   MachineConfig[11]."Unknown"."EM - 463"."PIT463-1".CW.ENABLE := True;

   MachineConfig[11]."Unit Sep"."EM - 400"."FIT409-1".CW.ENABLE := True;

   MachineConfig[11]."Unit Process"."EM - 201"."FCV201-1".CW.EXIST := False;

   MachineConfig[11]."Unit Process"."EM - 22X"."PCV22X-1".CW.NO := True;

   MachineConfig[11]."Unit Process"."EM - 22Y"."PCV22Y-1".CW.EXIST := False;

   MachineConfig[11]."Unit Sep"."EM - 400"."FCV409-1".CW.ENABLE := True;

   MachineConfig[11]."Unit Sep"."EM - 100".UPS.CW.EXIST := True;

   MachineConfig[11]."Unit Sep"."EM - 730".TS730.CW.ENABLE := True;

   MachineConfig[11]."Unit Dch"."EM - 222"."LS222-1".CW.EXIST := False;

   MachineConfig[11]."Unit Dch"."EM - 222"."P222-1".CW.EXIST := False;

   MachineConfig[11]."Unknown"."EM - 420"."P403-1".CW.EXIST := False;

   MachineConfig[11]."Unknown"."EM - 430"."P406-1".CW.EXIST := False;

   MachineConfig[11]."Unknown"."EM - 463"."P463-1".CW.ENABLE := True;

   MachineConfig[11]."Unknown"."EM - 463"."P463-1".CW.EXIST := False;

   MachineConfig[11]."Options"."EM - P201"."P201-1".CW.EXIST := False;

   MachineConfig[11]."Unknown"."EM - 208"."P208-1".CW.EXIST := False;

   MachineConfig[11]."Unit Sep"."EM - 100"."CA ERROR".CW.NO := True;

   MachineConfig[11]."Unit Sep"."EM - 100"."CA WD".CW.NO := True;

   MachineConfig[11]."Unit Sep"."EM - 400"."FIS412-1".CW.EXIST := False;

   MachineConfig[11]."Unknown"."EM - 420".LS422a.CW.EXIST := False;

   MachineConfig[11]."Unknown"."EM - 420"."LS42X(b)".CW.EXIST := False;

   MachineConfig[11]."Unknown"."EM - 420"."LS422-1".CW.EXIST := False;

   MachineConfig[11]."Unit Sep"."EM - 400"."FIT412-1".CW.EXIST := False;

   MachineConfig[11]."Unit Dch"."EM - 375"."PT37X-1".CW.ENABLE := True;

   MachineConfig[11]."Unit Dch"."EM - 375"."PT37X-1".CW.EXIST := False;

   MachineConfig[11]."Unit Dch"."EM - 222"."TT222-1".CW.ENABLE := True;

   MachineConfig[11]."Unit Sep"."EM - 400"."TT411-1".CW.EXIST := False;

   MachineConfig[11]."Unit Sep"."EM - 730".TT730b.CW.EXIST := False;

   MachineConfig[11]."Unit Sep"."EM - 730".TT734.CW.EXIST := False;

   MachineConfig[11]."Unit Sep"."EM - 400"."TT41X-1".CW.ENABLE := True;

   MachineConfig[11]."Unit Dch"."EM - 300"."AV302-1".CW.EXIST := False;

   MachineConfig[11]."Unit Dch"."EM - 300"."AV303-1".CW.ENABLE := True;

   MachineConfig[11]."Unit Dch"."EM - 300"."AV304-1".CW.ENABLE := True;

   MachineConfig[11]."Unit Dch"."EM - 300"."AV305-1".CW.ENABLE := True;

   MachineConfig[11]."Unit Dch"."EM - 300"."AV306-1".CW.EXIST := False;

   MachineConfig[11]."Unit Sep"."EM - 600"."AV615-1".CW.ENABLE := True;

   MachineConfig[11]."Unit Dch"."EM - 300"."AV635-1".CW.ENABLE := True;

   MachineConfig[11]."Unit Sep"."EM - 600"."AV63X/441-1".CW.EXIST := False;

   MachineConfig[11]."Unknown"."EM - 420"."PV421-1".CW.EXIST := False;

   MachineConfig[11]."Unknown"."EM - 420"."P421-1".CW.EXIST := False;

   MachineConfig[11]."Unit Dch"."EM - 506"."PV376-1".CW.ENABLE := True;

   MachineConfig[11]."Unit Dch"."EM - 506"."PV376-1".CW.EXIST := False;

   MachineConfig[11]."Unit Dch"."EM - 506"."PV376-2".CW.ENABLE := True;

   MachineConfig[11]."Unit Dch"."EM - 506"."PV376-2".CW.EXIST := False;

   MachineConfig[11]."Unit Dch"."EM - 506"."PV376-2".CW.NO := True;

   MachineConfig[11]."Unknown"."EM - 463"."AV660-1".CW.ENABLE := True;

   MachineConfig[11]."Unknown"."EM - 463"."AV660-1".CW.EXIST := False;

   MachineConfig[11]."Unknown"."EM - 463"."AV470-1".CW.ENABLE := True;

   MachineConfig[11]."Unknown"."EM - 463"."AV470-1".CW.EXIST := False;

   MachineConfig[11]."Unknown"."EM - 430"."AV430-1".CW.EXIST := False;

   MachineConfig[11]."Unknown"."EM - 463"."AV305-2".CW.ENABLE := True;

   MachineConfig[11]."Unknown"."EM - 463"."AV305-2".CW.EXIST := False;

   MachineConfig[11]."Unknown"."EM - 463"."AV660-2".CW.ENABLE := True;

   MachineConfig[11]."Unknown"."EM - 463"."AV660-2".CW.EXIST := False;

   MachineConfig[11]."Unit Process"."EM - 22Y"."FIT22Y-1".CW.EXIST := False;

   MachineConfig[12].Machine."Family" := 2;
   MachineConfig[12].Machine.TypeNo := 32;
   MachineConfig[12].Machine.Range := 1;
   MachineConfig[12].Machine.SepType := 1;
   MachineConfig[12].Machine.Frame := 1;
   MachineConfig[12].Machine.DchSystem := 2;
   MachineConfig[12].Machine.Spare_1 := 2;
   MachineConfig[12].Machine.FeedPump := 1;
   MachineConfig[12].Machine.Spare_2 := 2;
   MachineConfig[12].Machine.eMotion := 1;
   MachineConfig[12].Machine.ConditionAlert := 1;
   MachineConfig[12].Machine.eWON := 1;
   MachineConfig[12]."Unit Sep"."EM - 400"."TT41X-1".Address := 142;
   MachineConfig[12]."Unit Process"."EM - 201"."FIT201-1"."Type" := 2;
   MachineConfig[12]."Unit Process"."EM - 201"."FIT201-1".Address := 256;
   MachineConfig[12]."Unit Process"."EM - 201"."FIT201-1".Max := 65000.0;
   MachineConfig[12]."Unit Process"."EM - 22X"."FIT22X-1".Address := 276;
   MachineConfig[12]."Unit Process"."EM - 22X"."QT220-1".Tag := 'QT220-1';
   // === CW auto-patched for MachineConfig[12] ===

   MachineConfig[12]."Unknown"."EM - 208"."AV208-1".CW.VLV_W_FB := False;

   MachineConfig[12]."Unknown"."EM - 208"."AV208-1".CW.FB_OPN_EN := False;

   MachineConfig[12]."Unknown"."EM - 208"."AV208-1".CW.FB_CLS_EN := False;

   MachineConfig[12]."Unknown"."EM - 210"."AV210-1".CW.EXIST := False;

   MachineConfig[12]."Unknown"."EM - 210"."AV210-1".CW.VLV_W_FB := False;

   MachineConfig[12]."Unknown"."EM - 210"."AV210-1".CW.FB_OPN_EN := False;

   MachineConfig[12]."Unknown"."EM - 210"."AV210-1".CW.FB_CLS_EN := False;

   MachineConfig[12]."Unknown"."EM - 212"."AV212-1".CW.EXIST := False;

   MachineConfig[12]."Unknown"."EM - 212"."AV212-1".CW.VLV_W_FB := False;

   MachineConfig[12]."Unknown"."EM - 212"."AV212-1".CW.FB_OPN_EN := False;

   MachineConfig[12]."Unknown"."EM - 212"."AV212-1".CW.FB_CLS_EN := False;

   MachineConfig[12]."Unit Process"."EM - 22X"."AV220-1".CW.ENABLE := True;

   MachineConfig[12]."Unit Process"."EM - 22Y"."AV221-1".CW.EXIST := False;

   MachineConfig[12]."Unit Process"."EM - 22Y"."AV221-1".CW.VLV_W_FB := False;

   MachineConfig[12]."Unit Process"."EM - 22Y"."AV221-1".CW.FB_OPN_EN := False;

   MachineConfig[12]."Unit Process"."EM - 22Y"."AV221-1".CW.FB_CLS_EN := False;

   MachineConfig[12]."Unit Dch"."EM - 222"."AV222-1".CW.EXIST := False;

   MachineConfig[12]."Unit Dch"."EM - 222"."AV222-1".CW.VLV_W_FB := False;

   MachineConfig[12]."Unit Dch"."EM - 222"."AV222-1".CW.FB_OPN_EN := False;

   MachineConfig[12]."Unit Dch"."EM - 222"."AV222-1".CW.FB_CLS_EN := False;

   MachineConfig[12]."Unit Dch"."EM - 300"."AV320-1".CW.ENABLE := True;

   MachineConfig[12]."Unit Process"."EM - 340"."AV340-2".CW.ENABLE := True;

   MachineConfig[12]."Unit Process"."EM - 22X"."AV460-1".CW.ENABLE := True;

   MachineConfig[12]."Unit Process"."EM - 340"."AV460-2".CW.ENABLE := True;

   MachineConfig[12]."Unknown"."EM - 460"."AV460d-1".CW.EXIST := False;

   MachineConfig[12]."Unknown"."EM - 460"."AV460d-1".CW.VLV_W_FB := False;

   MachineConfig[12]."Unknown"."EM - 460"."AV460d-1".CW.FB_OPN_EN := False;

   MachineConfig[12]."Unknown"."EM - 460"."AV460d-1".CW.FB_CLS_EN := False;

   MachineConfig[12]."Unit Dch"."EM - 506"."AV543-1".CW.EXIST := False;

   MachineConfig[12]."Unit Dch"."EM - 506"."AV543-1".CW.VLV_W_FB := False;

   MachineConfig[12]."Unit Dch"."EM - 506"."AV543-1".CW.FB_OPN_EN := False;

   MachineConfig[12]."Unit Dch"."EM - 506"."AV543-1".CW.FB_CLS_EN := False;

   MachineConfig[12]."Unknown"."EM - 463"."AV463-1".CW.ENABLE := True;

   MachineConfig[12]."Unknown"."EM - 463"."AV463-1".CW.EXIST := False;

   MachineConfig[12]."Unknown"."EM - 463"."AV463-2".CW.ENABLE := True;

   MachineConfig[12]."Unknown"."EM - 463"."AV463-2".CW.EXIST := False;

   MachineConfig[12]."Unit Process"."EM - 22Y"."AV461-1".CW.EXIST := False;

   MachineConfig[12]."Unit Process"."EM - 22Y"."AV461-1".CW.VLV_W_FB := False;

   MachineConfig[12]."Unit Process"."EM - 22Y"."AV461-1".CW.FB_OPN_EN := False;

   MachineConfig[12]."Unit Process"."EM - 22Y"."AV461-1".CW.FB_CLS_EN := False;

   MachineConfig[12]."Unit Sep"."EM - 600"."FIS615-1".CW.ENABLE := True;

   MachineConfig[12]."Unit Sep"."EM - 600"."FIS635-1".CW.ENABLE := True;

   MachineConfig[12]."Unit Sep"."EM - 600"."FIS630-1".CW.EXIST := False;

   MachineConfig[12]."Unit Process"."EM - 340"."PIS340-1".CW.ENABLE := True;

   MachineConfig[12]."Unit Process"."EM - 201"."QT201-1_OK".CW.ENABLE := True;

   MachineConfig[12]."Unit Process"."EM - 22X"."QT220-1_OK".CW.ENABLE := True;

   MachineConfig[12]."Unit Process"."EM - 22X"."QT220-1_OK".CW.EXIST := False;

   MachineConfig[12]."Unit Process"."EM - 201"."LA201-1".CW.ENABLE := False;

   MachineConfig[12]."Unit Process"."EM - 201"."LA201-1".CW.EXIST := False;

   MachineConfig[12]."Unit Process"."EM - 22X"."LA220-1".CW.ENABLE := True;

   MachineConfig[12]."Unit Sep"."EM - 100"."L-GREEN".CW.ENABLE := True;

   MachineConfig[12]."Unit Sep"."EM - 100"."L-YELLOW".CW.EXIST := False;

   MachineConfig[12]."Unit Process"."EM - 22Y"."LA221-1".CW.EXIST := False;

   MachineConfig[12]."Unit Process"."EM - 201"."QT201-1".CW.ENABLE := True;

   MachineConfig[12]."Unit Process"."EM - 22X"."QT220-1".CW.ENABLE := True;

   MachineConfig[12]."Unit Process"."EM - 22X"."QT220-1".CW.EXIST := False;

   MachineConfig[12]."Unit Process"."EM - 22Y"."PIT22Y-1".CW.EXIST := False;

   MachineConfig[12]."Unknown"."EM - 463"."LT463-1".CW.ENABLE := True;

   MachineConfig[12]."Unknown"."EM - 463"."PIT463-1".CW.ENABLE := True;

   MachineConfig[12]."Unit Sep"."EM - 400"."FIT409-1".CW.ENABLE := True;

   MachineConfig[12]."Unit Process"."EM - 201"."FCV201-1".CW.EXIST := False;

   MachineConfig[12]."Unit Process"."EM - 22X"."PCV22X-1".CW.NO := True;

   MachineConfig[12]."Unit Process"."EM - 22Y"."PCV22Y-1".CW.EXIST := False;

   MachineConfig[12]."Unit Sep"."EM - 400"."FCV409-1".CW.ENABLE := True;

   MachineConfig[12]."Unit Sep"."EM - 100".UPS.CW.EXIST := True;

   MachineConfig[12]."Unit Sep"."EM - 730".TS730.CW.ENABLE := True;

   MachineConfig[12]."Unit Dch"."EM - 222"."LS222-1".CW.EXIST := False;

   MachineConfig[12]."Unit Dch"."EM - 222"."P222-1".CW.EXIST := False;

   MachineConfig[12]."Unknown"."EM - 420"."P403-1".CW.EXIST := False;

   MachineConfig[12]."Unknown"."EM - 430"."P406-1".CW.EXIST := False;

   MachineConfig[12]."Unknown"."EM - 463"."P463-1".CW.ENABLE := True;

   MachineConfig[12]."Unknown"."EM - 463"."P463-1".CW.EXIST := False;

   MachineConfig[12]."Options"."EM - P201"."P201-1".CW.EXIST := False;

   MachineConfig[12]."Unknown"."EM - 208"."P208-1".CW.EXIST := False;

   MachineConfig[12]."Unit Sep"."EM - 100"."CA VIB WARN".CW.ENABLE := True;

   MachineConfig[12]."Unit Sep"."EM - 100"."CA VIB WARN".CW.EXIST := True;

   MachineConfig[12]."Unit Sep"."EM - 100"."CA VIB ALM".CW.ENABLE := True;

   MachineConfig[12]."Unit Sep"."EM - 100"."CA VIB ALM".CW.EXIST := True;

   MachineConfig[12]."Unit Sep"."EM - 100"."CA ERROR".CW.ENABLE := True;

   MachineConfig[12]."Unit Sep"."EM - 100"."CA ERROR".CW.EXIST := True;

   MachineConfig[12]."Unit Sep"."EM - 100"."CA ERROR".CW.NO := True;

   MachineConfig[12]."Unit Sep"."EM - 100"."CA WD".CW.ENABLE := True;

   MachineConfig[12]."Unit Sep"."EM - 100"."CA WD".CW.EXIST := True;

   MachineConfig[12]."Unit Sep"."EM - 100"."CA WD".CW.NO := True;

   MachineConfig[12]."Unit Sep"."EM - 400"."FIS412-1".CW.EXIST := False;

   MachineConfig[12]."Unknown"."EM - 420".LS422a.CW.EXIST := False;

   MachineConfig[12]."Unknown"."EM - 420"."LS42X(b)".CW.EXIST := False;

   MachineConfig[12]."Unknown"."EM - 420"."LS422-1".CW.EXIST := False;

   MachineConfig[12]."Unit Sep"."EM - 400"."FIT412-1".CW.EXIST := False;

   MachineConfig[12]."Unit Dch"."EM - 375"."PT37X-1".CW.ENABLE := True;

   MachineConfig[12]."Unit Dch"."EM - 375"."PT37X-1".CW.EXIST := False;

   MachineConfig[12]."Unit Dch"."EM - 222"."TT222-1".CW.ENABLE := True;

   MachineConfig[12]."Unit Sep"."EM - 400"."TT411-1".CW.EXIST := False;

   MachineConfig[12]."Unit Sep"."EM - 730".TT730b.CW.EXIST := False;

   MachineConfig[12]."Unit Sep"."EM - 730".TT734.CW.EXIST := False;

   MachineConfig[12]."Unit Sep"."EM - 400"."TT41X-1".CW.ENABLE := True;

   MachineConfig[12]."Unit Dch"."EM - 300"."AV302-1".CW.ENABLE := True;

   MachineConfig[12]."Unit Dch"."EM - 300"."AV303-1".CW.ENABLE := True;

   MachineConfig[12]."Unit Dch"."EM - 300"."AV304-1".CW.ENABLE := True;

   MachineConfig[12]."Unit Dch"."EM - 300"."AV305-1".CW.ENABLE := True;

   MachineConfig[12]."Unit Dch"."EM - 300"."AV306-1".CW.EXIST := False;

   MachineConfig[12]."Unit Sep"."EM - 600"."AV615-1".CW.ENABLE := True;

   MachineConfig[12]."Unit Dch"."EM - 300"."AV635-1".CW.ENABLE := True;

   MachineConfig[12]."Unit Sep"."EM - 600"."AV63X/441-1".CW.EXIST := False;

   MachineConfig[12]."Unknown"."EM - 420"."PV421-1".CW.EXIST := False;

   MachineConfig[12]."Unknown"."EM - 420"."P421-1".CW.EXIST := False;

   MachineConfig[12]."Unit Dch"."EM - 506"."PV376-1".CW.ENABLE := True;

   MachineConfig[12]."Unit Dch"."EM - 506"."PV376-1".CW.EXIST := False;

   MachineConfig[12]."Unit Dch"."EM - 506"."PV376-2".CW.ENABLE := True;

   MachineConfig[12]."Unit Dch"."EM - 506"."PV376-2".CW.EXIST := False;

   MachineConfig[12]."Unit Dch"."EM - 506"."PV376-2".CW.NO := True;

   MachineConfig[12]."Unknown"."EM - 463"."AV660-1".CW.ENABLE := True;

   MachineConfig[12]."Unknown"."EM - 463"."AV660-1".CW.EXIST := False;

   MachineConfig[12]."Unknown"."EM - 463"."AV470-1".CW.ENABLE := True;

   MachineConfig[12]."Unknown"."EM - 463"."AV470-1".CW.EXIST := False;

   MachineConfig[12]."Unknown"."EM - 430"."AV430-1".CW.EXIST := False;

   MachineConfig[12]."Unknown"."EM - 463"."AV305-2".CW.ENABLE := True;

   MachineConfig[12]."Unknown"."EM - 463"."AV305-2".CW.EXIST := False;

   MachineConfig[12]."Unknown"."EM - 463"."AV660-2".CW.ENABLE := True;

   MachineConfig[12]."Unknown"."EM - 463"."AV660-2".CW.EXIST := False;

   MachineConfig[12]."Unit Process"."EM - 22Y"."FIT22Y-1".CW.EXIST := False;

   MachineConfig[13].Machine."Family" := 2;
   MachineConfig[13].Machine.TypeNo := 33;
   MachineConfig[13].Machine.Range := 1;
   MachineConfig[13].Machine.SepType := 1;
   MachineConfig[13].Machine.Frame := 1;
   MachineConfig[13].Machine.DchSystem := 2;
   MachineConfig[13].Machine.Spare_1 := 2;
   MachineConfig[13].Machine.FeedPump := 1;
   MachineConfig[13].Machine.Spare_2 := 2;
   MachineConfig[13].Machine.ConditionAlert := 1;
   MachineConfig[13].Machine.eWON := 1;
   MachineConfig[13]."Unit Sep"."EM - 400"."TT41X-1".Address := 142;
   MachineConfig[13]."Unit Sep"."EM - 600"."AV63X/441-1".TAG := 'AV441-1';
   MachineConfig[13]."Unit Sep"."EM - 600"."AV63X/441-1".ACT_OUT_ADD := 331;
   MachineConfig[13]."Unit Process"."EM - 201"."FIT201-1"."Type" := 2;
   MachineConfig[13]."Unit Process"."EM - 201"."FIT201-1".Address := 256;
   MachineConfig[13]."Unit Process"."EM - 201"."FIT201-1".Max := 65000.0;
   MachineConfig[13]."Unit Process"."EM - 22X"."FIT22X-1".Address := 276;
   MachineConfig[13]."Unit Process"."EM - 22X"."QT220-1".Tag := 'QT220-1';
   MachineConfig[13]."Unit Dch"."EM - 300"."AV635-1".TAG := 'AV441-1';
   // === CW auto-patched for MachineConfig[13] ===

   MachineConfig[13]."Unknown"."EM - 208"."AV208-1".CW.VLV_W_FB := False;

   MachineConfig[13]."Unknown"."EM - 208"."AV208-1".CW.FB_OPN_EN := False;

   MachineConfig[13]."Unknown"."EM - 208"."AV208-1".CW.FB_CLS_EN := False;

   MachineConfig[13]."Unknown"."EM - 210"."AV210-1".CW.EXIST := False;

   MachineConfig[13]."Unknown"."EM - 210"."AV210-1".CW.VLV_W_FB := False;

   MachineConfig[13]."Unknown"."EM - 210"."AV210-1".CW.FB_OPN_EN := False;

   MachineConfig[13]."Unknown"."EM - 210"."AV210-1".CW.FB_CLS_EN := False;

   MachineConfig[13]."Unknown"."EM - 212"."AV212-1".CW.EXIST := False;

   MachineConfig[13]."Unknown"."EM - 212"."AV212-1".CW.VLV_W_FB := False;

   MachineConfig[13]."Unknown"."EM - 212"."AV212-1".CW.FB_OPN_EN := False;

   MachineConfig[13]."Unknown"."EM - 212"."AV212-1".CW.FB_CLS_EN := False;

   MachineConfig[13]."Unit Process"."EM - 22X"."AV220-1".CW.ENABLE := True;

   MachineConfig[13]."Unit Process"."EM - 22Y"."AV221-1".CW.EXIST := False;

   MachineConfig[13]."Unit Process"."EM - 22Y"."AV221-1".CW.VLV_W_FB := False;

   MachineConfig[13]."Unit Process"."EM - 22Y"."AV221-1".CW.FB_OPN_EN := False;

   MachineConfig[13]."Unit Process"."EM - 22Y"."AV221-1".CW.FB_CLS_EN := False;

   MachineConfig[13]."Unit Dch"."EM - 222"."AV222-1".CW.EXIST := False;

   MachineConfig[13]."Unit Dch"."EM - 222"."AV222-1".CW.VLV_W_FB := False;

   MachineConfig[13]."Unit Dch"."EM - 222"."AV222-1".CW.FB_OPN_EN := False;

   MachineConfig[13]."Unit Dch"."EM - 222"."AV222-1".CW.FB_CLS_EN := False;

   MachineConfig[13]."Unit Dch"."EM - 300"."AV320-1".CW.ENABLE := True;

   MachineConfig[13]."Unit Process"."EM - 340"."AV340-2".CW.ENABLE := True;

   MachineConfig[13]."Unit Process"."EM - 22X"."AV460-1".CW.ENABLE := True;

   MachineConfig[13]."Unit Process"."EM - 340"."AV460-2".CW.ENABLE := True;

   MachineConfig[13]."Unknown"."EM - 460"."AV460d-1".CW.EXIST := False;

   MachineConfig[13]."Unknown"."EM - 460"."AV460d-1".CW.VLV_W_FB := False;

   MachineConfig[13]."Unknown"."EM - 460"."AV460d-1".CW.FB_OPN_EN := False;

   MachineConfig[13]."Unknown"."EM - 460"."AV460d-1".CW.FB_CLS_EN := False;

   MachineConfig[13]."Unit Dch"."EM - 506"."AV543-1".CW.EXIST := False;

   MachineConfig[13]."Unit Dch"."EM - 506"."AV543-1".CW.VLV_W_FB := False;

   MachineConfig[13]."Unit Dch"."EM - 506"."AV543-1".CW.FB_OPN_EN := False;

   MachineConfig[13]."Unit Dch"."EM - 506"."AV543-1".CW.FB_CLS_EN := False;

   MachineConfig[13]."Unknown"."EM - 463"."AV463-1".CW.EXIST := False;

   MachineConfig[13]."Unknown"."EM - 463"."AV463-1".CW.VLV_W_FB := False;

   MachineConfig[13]."Unknown"."EM - 463"."AV463-1".CW.FB_OPN_EN := False;

   MachineConfig[13]."Unknown"."EM - 463"."AV463-1".CW.FB_CLS_EN := False;

   MachineConfig[13]."Unknown"."EM - 463"."AV463-2".CW.EXIST := False;

   MachineConfig[13]."Unknown"."EM - 463"."AV463-2".CW.VLV_W_FB := False;

   MachineConfig[13]."Unknown"."EM - 463"."AV463-2".CW.FB_OPN_EN := False;

   MachineConfig[13]."Unknown"."EM - 463"."AV463-2".CW.FB_CLS_EN := False;

   MachineConfig[13]."Unit Process"."EM - 22Y"."AV461-1".CW.EXIST := False;

   MachineConfig[13]."Unit Process"."EM - 22Y"."AV461-1".CW.VLV_W_FB := False;

   MachineConfig[13]."Unit Process"."EM - 22Y"."AV461-1".CW.FB_OPN_EN := False;

   MachineConfig[13]."Unit Process"."EM - 22Y"."AV461-1".CW.FB_CLS_EN := False;

   MachineConfig[13]."Unit Sep"."EM - 600"."FIS615-1".CW.ENABLE := True;

   MachineConfig[13]."Unit Sep"."EM - 600"."FIS635-1".CW.ENABLE := True;

   MachineConfig[13]."Unit Sep"."EM - 600"."FIS630-1".CW.EXIST := False;

   MachineConfig[13]."Unit Process"."EM - 340"."PIS340-1".CW.ENABLE := True;

   MachineConfig[13]."Unit Process"."EM - 201"."QT201-1_OK".CW.ENABLE := True;

   MachineConfig[13]."Unit Process"."EM - 22X"."QT220-1_OK".CW.ENABLE := True;

   MachineConfig[13]."Unit Process"."EM - 22X"."QT220-1_OK".CW.EXIST := False;

   MachineConfig[13]."Unit Process"."EM - 201"."LA201-1".CW.ENABLE := False;

   MachineConfig[13]."Unit Process"."EM - 201"."LA201-1".CW.EXIST := False;

   MachineConfig[13]."Unit Process"."EM - 22X"."LA220-1".CW.ENABLE := True;

   MachineConfig[13]."Unit Sep"."EM - 100"."L-GREEN".CW.ENABLE := True;

   MachineConfig[13]."Unit Sep"."EM - 100"."L-YELLOW".CW.EXIST := False;

   MachineConfig[13]."Unit Process"."EM - 22Y"."LA221-1".CW.EXIST := False;

   MachineConfig[13]."Unit Process"."EM - 201"."QT201-1".CW.ENABLE := True;

   MachineConfig[13]."Unit Process"."EM - 22X"."QT220-1".CW.ENABLE := True;

   MachineConfig[13]."Unit Process"."EM - 22X"."QT220-1".CW.EXIST := False;

   MachineConfig[13]."Unit Process"."EM - 22Y"."PIT22Y-1".CW.EXIST := False;

   MachineConfig[13]."Unit Sep"."EM - 400"."FIT409-1".CW.ENABLE := True;

   MachineConfig[13]."Unit Process"."EM - 201"."FCV201-1".CW.EXIST := False;

   MachineConfig[13]."Unit Process"."EM - 22X"."PCV22X-1".CW.NO := True;

   MachineConfig[13]."Unit Process"."EM - 22Y"."PCV22Y-1".CW.EXIST := False;

   MachineConfig[13]."Unit Sep"."EM - 400"."FCV409-1".CW.ENABLE := True;

   MachineConfig[13]."Unit Sep"."EM - 100".UPS.CW.EXIST := True;

   MachineConfig[13]."Unit Sep"."EM - 730".TS730.CW.ENABLE := True;

   MachineConfig[13]."Unit Dch"."EM - 222"."LS222-1".CW.EXIST := False;

   MachineConfig[13]."Unit Dch"."EM - 222"."P222-1".CW.EXIST := False;

   MachineConfig[13]."Unknown"."EM - 420"."P403-1".CW.EXIST := False;

   MachineConfig[13]."Unknown"."EM - 430"."P406-1".CW.EXIST := False;

   MachineConfig[13]."Unknown"."EM - 463"."P463-1".CW.EXIST := False;

   MachineConfig[13]."Options"."EM - P201"."P201-1".CW.EXIST := False;

   MachineConfig[13]."Unknown"."EM - 208"."P208-1".CW.EXIST := False;

   MachineConfig[13]."Unit Sep"."EM - 100"."CA ERROR".CW.NO := True;

   MachineConfig[13]."Unit Sep"."EM - 100"."CA WD".CW.NO := True;

   MachineConfig[13]."Unit Sep"."EM - 400"."FIS412-1".CW.EXIST := False;

   MachineConfig[13]."Unknown"."EM - 420".LS422a.CW.EXIST := False;

   MachineConfig[13]."Unknown"."EM - 420"."LS42X(b)".CW.EXIST := False;

   MachineConfig[13]."Unknown"."EM - 420"."LS422-1".CW.EXIST := False;

   MachineConfig[13]."Unit Sep"."EM - 400"."FIT412-1".CW.EXIST := False;

   MachineConfig[13]."Unit Dch"."EM - 375"."PT37X-1".CW.EXIST := False;

   MachineConfig[13]."Unit Dch"."EM - 222"."TT222-1".CW.ENABLE := True;

   MachineConfig[13]."Unit Sep"."EM - 400"."TT411-1".CW.EXIST := False;

   MachineConfig[13]."Unit Sep"."EM - 730".TT730b.CW.EXIST := False;

   MachineConfig[13]."Unit Sep"."EM - 730".TT734.CW.EXIST := False;

   MachineConfig[13]."Unit Sep"."EM - 400"."TT41X-1".CW.ENABLE := True;

   MachineConfig[13]."Unit Dch"."EM - 300"."AV302-1".CW.EXIST := False;

   MachineConfig[13]."Unit Dch"."EM - 300"."AV303-1".CW.ENABLE := True;

   MachineConfig[13]."Unit Dch"."EM - 300"."AV304-1".CW.ENABLE := True;

   MachineConfig[13]."Unit Dch"."EM - 300"."AV305-1".CW.ENABLE := True;

   MachineConfig[13]."Unit Dch"."EM - 300"."AV306-1".CW.EXIST := False;

   MachineConfig[13]."Unit Sep"."EM - 600"."AV615-1".CW.ENABLE := True;

   MachineConfig[13]."Unit Dch"."EM - 300"."AV635-1".CW.ENABLE := True;

   MachineConfig[13]."Unit Sep"."EM - 600"."AV63X/441-1".CW.EXIST := False;

   MachineConfig[13]."Unknown"."EM - 420"."PV421-1".CW.EXIST := False;

   MachineConfig[13]."Unknown"."EM - 420"."P421-1".CW.EXIST := False;

   MachineConfig[13]."Unit Dch"."EM - 506"."PV376-1".CW.EXIST := False;

   MachineConfig[13]."Unit Dch"."EM - 506"."PV376-2".CW.EXIST := False;

   MachineConfig[13]."Unit Dch"."EM - 506"."PV376-2".CW.NO := True;

   MachineConfig[13]."Unknown"."EM - 463"."AV660-1".CW.EXIST := False;

   MachineConfig[13]."Unknown"."EM - 463"."AV470-1".CW.EXIST := False;

   MachineConfig[13]."Unknown"."EM - 430"."AV430-1".CW.EXIST := False;

   MachineConfig[13]."Unknown"."EM - 463"."AV305-2".CW.EXIST := False;

   MachineConfig[13]."Unknown"."EM - 463"."AV660-2".CW.EXIST := False;

   MachineConfig[13]."Unit Process"."EM - 22Y"."FIT22Y-1".CW.EXIST := False;

   MachineConfig[14].Machine."Family" := 2;
   MachineConfig[14].Machine.TypeNo := 34;
   MachineConfig[14].Machine.Range := 1;
   MachineConfig[14].Machine.SepType := 1;
   MachineConfig[14].Machine.Frame := 1;
   MachineConfig[14].Machine.DchSystem := 2;
   MachineConfig[14].Machine.Spare_1 := 2;
   MachineConfig[14].Machine.FeedPump := 1;
   MachineConfig[14].Machine.Spare_2 := 2;
   MachineConfig[14].Machine.eMotion := 1;
   MachineConfig[14].Machine.ConditionAlert := 1;
   MachineConfig[14].Machine.eWON := 1;
   MachineConfig[14]."Unit Sep"."EM - 400"."TT41X-1".Tag := 'TT410-1';
   MachineConfig[14]."Unit Sep"."EM - 600"."AV63X/441-1".TAG := 'AV635-1';
   MachineConfig[14]."Unit Process"."EM - 201"."FIT201-1"."Type" := 2;
   MachineConfig[14]."Unit Process"."EM - 201"."FIT201-1".Address := 256;
   MachineConfig[14]."Unit Process"."EM - 201"."FIT201-1".Max := 65000.0;
   MachineConfig[14]."Unit Process"."EM - 22X"."FIT22X-1".Address := 276;
   MachineConfig[14]."Unit Process"."EM - 22X"."QT220-1".Tag := 'QT220-1';
   MachineConfig[14]."Unit Process"."EM - 22X"."QT220-1".Address := 70;
   // === CW auto-patched for MachineConfig[14] ===

   MachineConfig[14]."Unknown"."EM - 208"."AV208-1".CW.VLV_W_FB := False;

   MachineConfig[14]."Unknown"."EM - 208"."AV208-1".CW.FB_OPN_EN := False;

   MachineConfig[14]."Unknown"."EM - 208"."AV208-1".CW.FB_CLS_EN := False;

   MachineConfig[14]."Unknown"."EM - 210"."AV210-1".CW.EXIST := False;

   MachineConfig[14]."Unknown"."EM - 210"."AV210-1".CW.VLV_W_FB := False;

   MachineConfig[14]."Unknown"."EM - 210"."AV210-1".CW.FB_OPN_EN := False;

   MachineConfig[14]."Unknown"."EM - 210"."AV210-1".CW.FB_CLS_EN := False;

   MachineConfig[14]."Unknown"."EM - 212"."AV212-1".CW.EXIST := False;

   MachineConfig[14]."Unknown"."EM - 212"."AV212-1".CW.VLV_W_FB := False;

   MachineConfig[14]."Unknown"."EM - 212"."AV212-1".CW.FB_OPN_EN := False;

   MachineConfig[14]."Unknown"."EM - 212"."AV212-1".CW.FB_CLS_EN := False;

   MachineConfig[14]."Unit Process"."EM - 22X"."AV220-1".CW.ENABLE := True;

   MachineConfig[14]."Unit Process"."EM - 22Y"."AV221-1".CW.EXIST := False;

   MachineConfig[14]."Unit Process"."EM - 22Y"."AV221-1".CW.VLV_W_FB := False;

   MachineConfig[14]."Unit Process"."EM - 22Y"."AV221-1".CW.FB_OPN_EN := False;

   MachineConfig[14]."Unit Process"."EM - 22Y"."AV221-1".CW.FB_CLS_EN := False;

   MachineConfig[14]."Unit Dch"."EM - 222"."AV222-1".CW.EXIST := False;

   MachineConfig[14]."Unit Dch"."EM - 222"."AV222-1".CW.VLV_W_FB := False;

   MachineConfig[14]."Unit Dch"."EM - 222"."AV222-1".CW.FB_OPN_EN := False;

   MachineConfig[14]."Unit Dch"."EM - 222"."AV222-1".CW.FB_CLS_EN := False;

   MachineConfig[14]."Unit Dch"."EM - 300"."AV320-1".CW.ENABLE := True;

   MachineConfig[14]."Unit Process"."EM - 340"."AV340-2".CW.ENABLE := True;

   MachineConfig[14]."Unit Process"."EM - 22X"."AV460-1".CW.ENABLE := True;

   MachineConfig[14]."Unit Process"."EM - 340"."AV460-2".CW.ENABLE := True;

   MachineConfig[14]."Unknown"."EM - 460"."AV460d-1".CW.EXIST := False;

   MachineConfig[14]."Unknown"."EM - 460"."AV460d-1".CW.VLV_W_FB := False;

   MachineConfig[14]."Unknown"."EM - 460"."AV460d-1".CW.FB_OPN_EN := False;

   MachineConfig[14]."Unknown"."EM - 460"."AV460d-1".CW.FB_CLS_EN := False;

   MachineConfig[14]."Unit Dch"."EM - 506"."AV543-1".CW.EXIST := False;

   MachineConfig[14]."Unit Dch"."EM - 506"."AV543-1".CW.VLV_W_FB := False;

   MachineConfig[14]."Unit Dch"."EM - 506"."AV543-1".CW.FB_OPN_EN := False;

   MachineConfig[14]."Unit Dch"."EM - 506"."AV543-1".CW.FB_CLS_EN := False;

   MachineConfig[14]."Unknown"."EM - 463"."AV463-1".CW.ENABLE := True;

   MachineConfig[14]."Unknown"."EM - 463"."AV463-1".CW.EXIST := False;

   MachineConfig[14]."Unknown"."EM - 463"."AV463-2".CW.ENABLE := True;

   MachineConfig[14]."Unknown"."EM - 463"."AV463-2".CW.EXIST := False;

   MachineConfig[14]."Unit Process"."EM - 22Y"."AV461-1".CW.EXIST := False;

   MachineConfig[14]."Unit Process"."EM - 22Y"."AV461-1".CW.VLV_W_FB := False;

   MachineConfig[14]."Unit Process"."EM - 22Y"."AV461-1".CW.FB_OPN_EN := False;

   MachineConfig[14]."Unit Process"."EM - 22Y"."AV461-1".CW.FB_CLS_EN := False;

   MachineConfig[14]."Unit Sep"."EM - 600"."FIS615-1".CW.ENABLE := True;

   MachineConfig[14]."Unit Sep"."EM - 600"."FIS635-1".CW.ENABLE := True;

   MachineConfig[14]."Unit Sep"."EM - 600"."FIS630-1".CW.EXIST := False;

   MachineConfig[14]."Unit Process"."EM - 340"."PIS340-1".CW.ENABLE := True;

   MachineConfig[14]."Unit Process"."EM - 201"."QT201-1_OK".CW.ENABLE := True;

   MachineConfig[14]."Unit Process"."EM - 22X"."QT220-1_OK".CW.ENABLE := True;

   MachineConfig[14]."Unit Process"."EM - 22X"."QT220-1_OK".CW.EXIST := False;

   MachineConfig[14]."Unit Process"."EM - 201"."LA201-1".CW.ENABLE := False;

   MachineConfig[14]."Unit Process"."EM - 201"."LA201-1".CW.EXIST := False;

   MachineConfig[14]."Unit Process"."EM - 22X"."LA220-1".CW.ENABLE := True;

   MachineConfig[14]."Unit Sep"."EM - 100"."L-GREEN".CW.ENABLE := True;

   MachineConfig[14]."Unit Sep"."EM - 100"."L-YELLOW".CW.EXIST := False;

   MachineConfig[14]."Unit Process"."EM - 22Y"."LA221-1".CW.EXIST := False;

   MachineConfig[14]."Unit Process"."EM - 201"."QT201-1".CW.ENABLE := True;

   MachineConfig[14]."Unit Process"."EM - 22X"."QT220-1".CW.ENABLE := True;

   MachineConfig[14]."Unit Process"."EM - 22X"."QT220-1".CW.EXIST := False;

   MachineConfig[14]."Unit Process"."EM - 22Y"."PIT22Y-1".CW.EXIST := False;

   MachineConfig[14]."Unknown"."EM - 463"."LT463-1".CW.ENABLE := True;

   MachineConfig[14]."Unknown"."EM - 463"."PIT463-1".CW.ENABLE := True;

   MachineConfig[14]."Unit Sep"."EM - 400"."FIT409-1".CW.ENABLE := True;

   MachineConfig[14]."Unit Process"."EM - 201"."FCV201-1".CW.EXIST := False;

   MachineConfig[14]."Unit Process"."EM - 22X"."PCV22X-1".CW.NO := True;

   MachineConfig[14]."Unit Process"."EM - 22Y"."PCV22Y-1".CW.EXIST := False;

   MachineConfig[14]."Unit Sep"."EM - 400"."FCV409-1".CW.ENABLE := True;

   MachineConfig[14]."Unit Sep"."EM - 100".UPS.CW.EXIST := True;

   MachineConfig[14]."Unit Sep"."EM - 730".TS730.CW.ENABLE := True;

   MachineConfig[14]."Unit Dch"."EM - 222"."LS222-1".CW.EXIST := False;

   MachineConfig[14]."Unit Dch"."EM - 222"."P222-1".CW.EXIST := False;

   MachineConfig[14]."Unknown"."EM - 420"."P403-1".CW.EXIST := False;

   MachineConfig[14]."Unknown"."EM - 430"."P406-1".CW.EXIST := False;

   MachineConfig[14]."Unknown"."EM - 463"."P463-1".CW.ENABLE := True;

   MachineConfig[14]."Unknown"."EM - 463"."P463-1".CW.EXIST := False;

   MachineConfig[14]."Options"."EM - P201"."P201-1".CW.EXIST := False;

   MachineConfig[14]."Unknown"."EM - 208"."P208-1".CW.EXIST := False;

   MachineConfig[14]."Unit Sep"."EM - 100"."CA VIB WARN".CW.ENABLE := True;

   MachineConfig[14]."Unit Sep"."EM - 100"."CA VIB WARN".CW.EXIST := True;

   MachineConfig[14]."Unit Sep"."EM - 100"."CA VIB ALM".CW.ENABLE := True;

   MachineConfig[14]."Unit Sep"."EM - 100"."CA VIB ALM".CW.EXIST := True;

   MachineConfig[14]."Unit Sep"."EM - 100"."CA ERROR".CW.ENABLE := True;

   MachineConfig[14]."Unit Sep"."EM - 100"."CA ERROR".CW.EXIST := True;

   MachineConfig[14]."Unit Sep"."EM - 100"."CA ERROR".CW.NO := True;

   MachineConfig[14]."Unit Sep"."EM - 100"."CA WD".CW.ENABLE := True;

   MachineConfig[14]."Unit Sep"."EM - 100"."CA WD".CW.EXIST := True;

   MachineConfig[14]."Unit Sep"."EM - 100"."CA WD".CW.NO := True;

   MachineConfig[14]."Unit Sep"."EM - 400"."FIS412-1".CW.EXIST := False;

   MachineConfig[14]."Unknown"."EM - 420".LS422a.CW.EXIST := False;

   MachineConfig[14]."Unknown"."EM - 420"."LS42X(b)".CW.EXIST := False;

   MachineConfig[14]."Unknown"."EM - 420"."LS422-1".CW.EXIST := False;

   MachineConfig[14]."Unit Sep"."EM - 400"."FIT412-1".CW.EXIST := False;

   MachineConfig[14]."Unit Dch"."EM - 375"."PT37X-1".CW.ENABLE := True;

   MachineConfig[14]."Unit Dch"."EM - 375"."PT37X-1".CW.EXIST := False;

   MachineConfig[14]."Unit Dch"."EM - 222"."TT222-1".CW.ENABLE := True;

   MachineConfig[14]."Unit Sep"."EM - 400"."TT411-1".CW.EXIST := False;

   MachineConfig[14]."Unit Sep"."EM - 730".TT730b.CW.EXIST := False;

   MachineConfig[14]."Unit Sep"."EM - 730".TT734.CW.EXIST := False;

   MachineConfig[14]."Unit Sep"."EM - 400"."TT41X-1".CW.ENABLE := True;

   MachineConfig[14]."Unit Dch"."EM - 300"."AV302-1".CW.ENABLE := True;

   MachineConfig[14]."Unit Dch"."EM - 300"."AV303-1".CW.ENABLE := True;

   MachineConfig[14]."Unit Dch"."EM - 300"."AV304-1".CW.ENABLE := True;

   MachineConfig[14]."Unit Dch"."EM - 300"."AV305-1".CW.ENABLE := True;

   MachineConfig[14]."Unit Dch"."EM - 300"."AV306-1".CW.EXIST := False;

   MachineConfig[14]."Unit Sep"."EM - 600"."AV615-1".CW.ENABLE := True;

   MachineConfig[14]."Unit Dch"."EM - 300"."AV635-1".CW.ENABLE := True;

   MachineConfig[14]."Unit Sep"."EM - 600"."AV63X/441-1".CW.EXIST := False;

   MachineConfig[14]."Unknown"."EM - 420"."PV421-1".CW.EXIST := False;

   MachineConfig[14]."Unknown"."EM - 420"."P421-1".CW.EXIST := False;

   MachineConfig[14]."Unit Dch"."EM - 506"."PV376-1".CW.ENABLE := True;

   MachineConfig[14]."Unit Dch"."EM - 506"."PV376-1".CW.EXIST := False;

   MachineConfig[14]."Unit Dch"."EM - 506"."PV376-2".CW.ENABLE := True;

   MachineConfig[14]."Unit Dch"."EM - 506"."PV376-2".CW.EXIST := False;

   MachineConfig[14]."Unit Dch"."EM - 506"."PV376-2".CW.NO := True;

   MachineConfig[14]."Unknown"."EM - 463"."AV660-1".CW.ENABLE := True;

   MachineConfig[14]."Unknown"."EM - 463"."AV660-1".CW.EXIST := False;

   MachineConfig[14]."Unknown"."EM - 463"."AV470-1".CW.ENABLE := True;

   MachineConfig[14]."Unknown"."EM - 463"."AV470-1".CW.EXIST := False;

   MachineConfig[14]."Unknown"."EM - 430"."AV430-1".CW.EXIST := False;

   MachineConfig[14]."Unknown"."EM - 463"."AV305-2".CW.ENABLE := True;

   MachineConfig[14]."Unknown"."EM - 463"."AV305-2".CW.EXIST := False;

   MachineConfig[14]."Unknown"."EM - 463"."AV660-2".CW.ENABLE := True;

   MachineConfig[14]."Unknown"."EM - 463"."AV660-2".CW.EXIST := False;

   MachineConfig[14]."Unit Process"."EM - 22Y"."FIT22Y-1".CW.EXIST := False;


END_DATA_BLOCK

